TYPE ST_ElementRegistryConv :
(**************************************************************************************
 * 	Application		:	BoxControl Framework
 *	Revision		:	$Revision: 404529 $
 *	Revision date	:	$Date: 2018-04-23 08:21:38 +0200 (Mo., 23 Apr 2018) $
 *	Last changed by	:	$Author: b7bolm $
 *	URL				:	$URL: http://almscdc.swisslog.com/repo/SWPD/Development/BoxControlFramework/20_Release/trunk/01_Software/BCF/BCF/JumpStart/20_Product/10_App/10_Base/10_Lib/10_Conv/01_DUTs/ST_ElementRegistryConv.TcDUT $
 *
 *	Purpose			:	Element registration structure.
 *
 * ------------------------------------------------------------------------------------
 *	Copyright Swisslog [IP AG], Switzerland. All rights reserved.
 * 
 * ------------------------------------------------------------------------------------
 *	
 * 	Revision History: 
 *
 * 	VERSION			DATE			INITIALS			DESCRIPTION
 *	0.1				01.01.2001		swl					Example
 *
 **************************************************************************************)
STRUCT
	Enable				: BOOL; // Element enabled 
	ElementName			: STRING(System.NAME_LENGTH); // Name as string
	eElementNumber		: E_ElementNumber; // Element number 
	eElementType		: E_ElementType; // Element type
	rElementData		: REFERENCE TO ST_ElementData; 
	rElementInterface 	: REFERENCE TO ST_ElementInterface;
	rSettingsElement	: REFERENCE TO ST_CFG_Element;
	rElement			: REFERENCE TO FB_ElementConv; // Reference to Element 
	HashCode			: UDINT; // HashCode
END_STRUCT
END_TYPE

(* stored: Version 1.1.0.1, ProductVersion 3.1.4022.12
   DUT ST_ElementRegistryConv: Id {25189a3e-78c6-4124-b37b-dd1fd61f6557} *)
